Staubli VAL3: Header.dtx

mdesc mNomSpeed
public num nMsgType
public num nCommType
public num nReplyCode
